TYPE ST_MainStateMachineHmiCommand :
STRUCT
	bStartButton				: BOOL;
	bStopButton					: BOOL;
END_STRUCT
END_TYPE

(* stored: Version 1.1.0.1, ProductVersion 3.1.4024.11
   DUT ST_MainStateMachineHmiCommand: Id {7dffa93f-dee1-42ca-b3b2-e08f9bf3a6ce} *)
